FUNCTION_BLOCK FB_Fan
VAR_INPUT
	bInputControl	:	BOOL;
	iTempIn			:	INT := 0;
	iTempOut		:	INT := 0;
END_VAR
VAR_IN_OUT
	bInputHA		:	BOOL;						//Input (HA)
END_VAR
VAR_OUTPUT
	bOut			:	BOOL;
END_VAR
VAR CONSTANT
END_VAR
VAR
	rTempIn			:	REAL;
	rTempOut		:	REAL;
	bTempLock		:	BOOL := FALSE;
END_VAR

IF bInputHA THEN

	bOut := TRUE;

ELSE

//	rTempIn		:= iTempIn 	/ 10;
//	rTempOut	:= iTempOut / 10;
	
//	IF (rTempOut < rTempIn) AND (rTempIn < 2) THEN
	
//		bTempLock	:=	TRUE;
	
//	ELSE
	
//		bTempLock	:= 	FALSE;
	
//	END_IF

	IF bTempLock THEN
		bOut	:= FALSE;
	ELSE
		bOut := bInputControl;
	END_IF

END_IF

END_FUNCTION_BLOCK

(* stored: Version 1.1.0.1, ProductVersion 3.1.4024.4
   POU FB_Fan: Id {682d3b5f-49e2-40c6-8dd2-030b9b586ca1}, SpecialFunc None *)
